FUNCTION_BLOCK DIV_LINT (* IEC 61131-3 LINT Division *)
  (* Standard: 61131-3 *)
  (* Version 0.0, 2004-12-15, JHC, Rockwell Automation, Converted from SRC format. *)
  (* Compiler header: package fb.rt.plc.math; *)
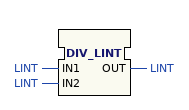
  VAR_INPUT
    IN1 : LINT; (* Dividend *)
    IN2 : LINT; (* Divisor *)
  END_VAR
  VAR_OUTPUT
    OUT : LINT; (* Quotient *)
  END_VAR
END_FUNCTION_BLOCK
